// TIA Portal V21 export
DATA_BLOCK "DTL"   // DB100
{ S7_Optimized_Access := 'TRUE' }
// stored: MemoryReserve 100
   VAR RETAIN
      READ : DTL;
      WRITE : DTL;
      "RET READ" : Int := 0;
      "RET WRITE" : Int := 0;
      SET : Bool := FALSE;
   END_VAR
BEGIN
END_DATA_BLOCK
